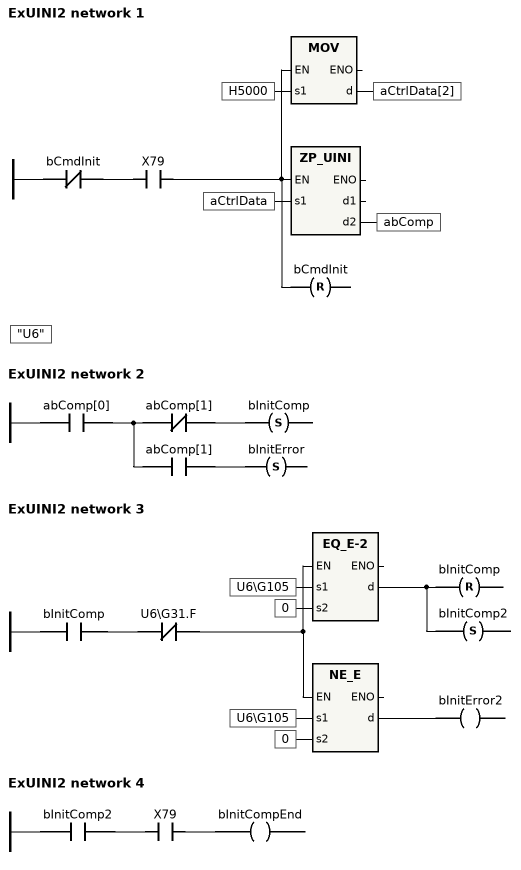
(* [picture p48: structured ladder/FBD of ExUINI2, networks 1 to 4] *)
(* network 1 *)
_p1 := NOT bCmdInit AND X79;
MOV(_p1, H5000, aCtrlData[2]);
ZP_UINI(_p1, aCtrlData, _open, abComp);
RST(_p1, bCmdInit);
(* not connected to any output: "U6" *)
(* network 2 *)
SET(abComp[0] AND NOT abComp[1], bInitComp);
SET(abComp[0] AND abComp[1], bInitError);
(* network 3 *)
_p1 := bInitComp AND NOT U6\G31.F;
EQ_E(_p1, U6\G105, 0, _t2);
RST(_t2, bInitComp);
SET(_t2, bInitComp2);
NE_E(_p1, U6\G105, 0, _t3);
bInitError2 := _t3;
(* network 4 *)
bInitCompEnd := bInitComp2 AND X79;
END_PROGRAM

PROGRAM ExEthSREAD_SWRITE
VAR
  Mov8INT_1 : Mov8INT;
  acRdCtrl : ARRAY [0..17] OF INT;
  abRdComp : ARRAY [0..1] OF BOOL;
  iCntRdOk : INT;
  iCntRdErr : INT;
  acWrCtrl : ARRAY [0..17] OF INT;
  abWrComp : ARRAY [0..1] OF BOOL;
  Mov8INT_2 : Mov8INT;
  iCntWrOk : INT;
  iCntWrErr : INT;
  bRdOK : BOOL;
  bWrOK : BOOL;
END_VAR
(* structured ladder/FBD written out as ST: instructions are called as NAME(EN, inputs, outputs); _pN, _eN, _tN stand for wires *)
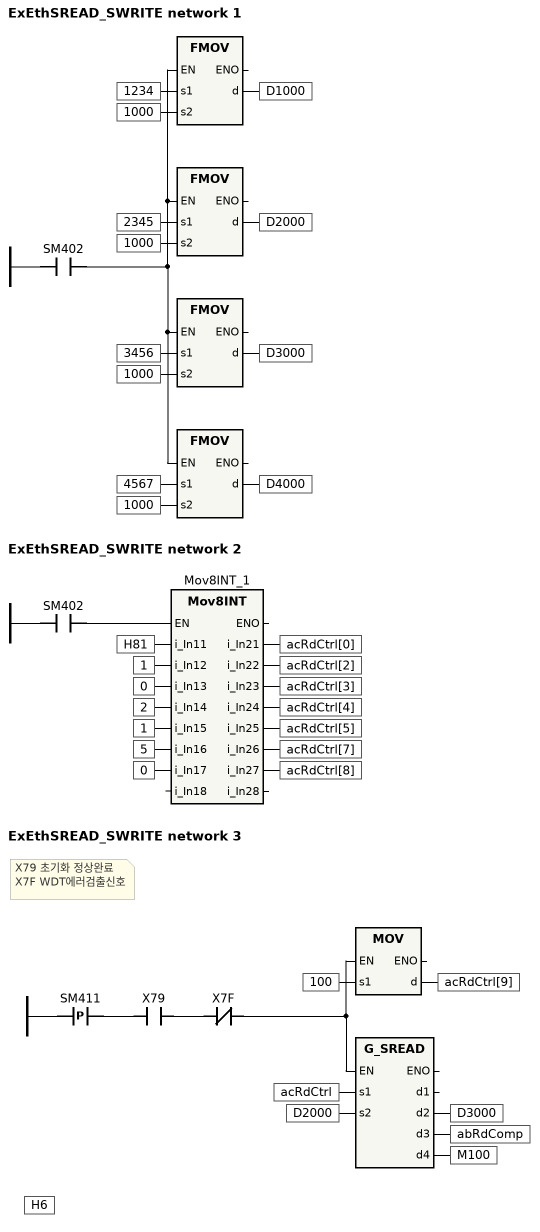
(* network 1 *)
FMOV(SM402, 1234, 1000, D1000);
FMOV(SM402, 2345, 1000, D2000);
FMOV(SM402, 3456, 1000, D3000);
FMOV(SM402, 4567, 1000, D4000);
(* network 2 *)
Mov8INT_1(EN := SM402, i_In11 := H81, i_In12 := 1, i_In13 := 0, i_In14 := 2, i_In15 := 1, i_In16 := 5, i_In17 := 0, i_In21 => acRdCtrl[0], i_In22 => acRdCtrl[2], i_In23 => acRdCtrl[3], i_In24 => acRdCtrl[4], i_In25 => acRdCtrl[5], i_In26 => acRdCtrl[7], i_In27 => acRdCtrl[8]);
(* network 3 *)
(* X79 초기화 정상완료 / X7F WDT에러검출신호 *)
_p1 := LDP(TRUE, SM411) AND X79 AND NOT X7F;
MOV(_p1, 100, acRdCtrl[9]);
G_SREAD(_p1, acRdCtrl, D2000, _open, D3000, abRdComp, M100);
(* not connected to any output: H6 *)
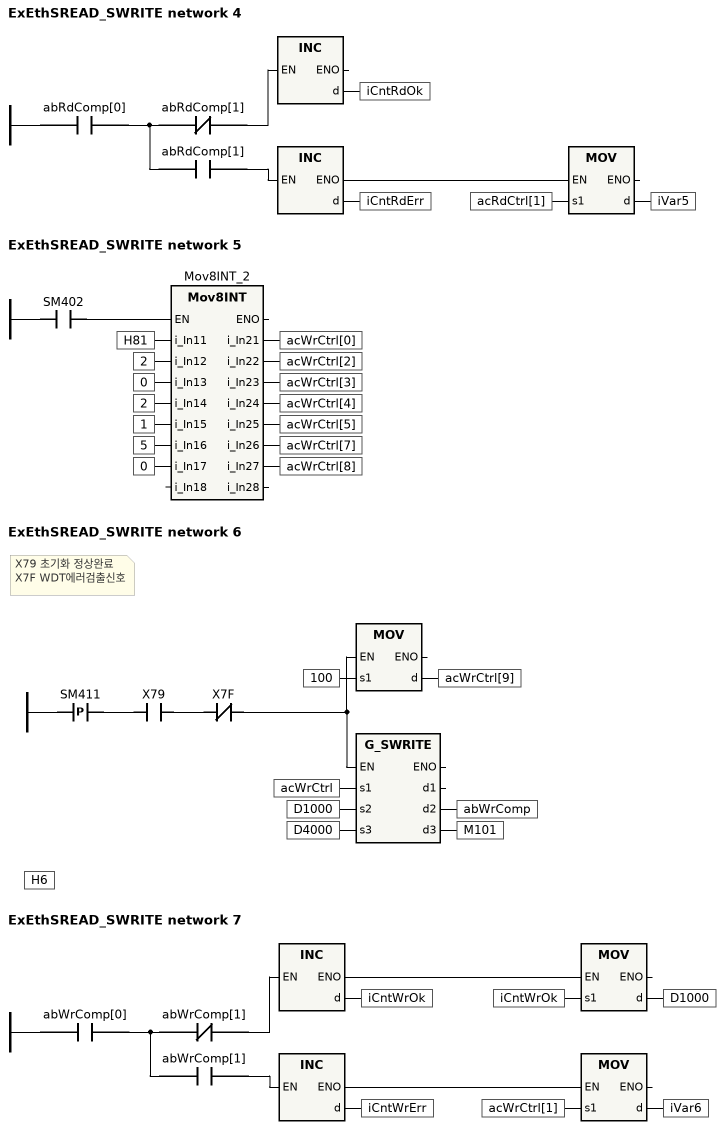
(* network 4 *)
INC(abRdComp[0] AND NOT abRdComp[1], iCntRdOk);
_e1 := INC(abRdComp[0] AND abRdComp[1], iCntRdErr);
MOV(_e1, acRdCtrl[1], iVar5);
(* network 5 *)
Mov8INT_2(EN := SM402, i_In11 := H81, i_In12 := 2, i_In13 := 0, i_In14 := 2, i_In15 := 1, i_In16 := 5, i_In17 := 0, i_In21 => acWrCtrl[0], i_In22 => acWrCtrl[2], i_In23 => acWrCtrl[3], i_In24 => acWrCtrl[4], i_In25 => acWrCtrl[5], i_In26 => acWrCtrl[7], i_In27 => acWrCtrl[8]);
(* network 6 *)
(* X79 초기화 정상완료 / X7F WDT에러검출신호 *)
_p1 := LDP(TRUE, SM411) AND X79 AND NOT X7F;
MOV(_p1, 100, acWrCtrl[9]);
G_SWRITE(_p1, acWrCtrl, D1000, D4000, _open, abWrComp, M101);
(* not connected to any output: H6 *)
(* network 7 *)
_e1 := INC(abWrComp[0] AND NOT abWrComp[1], iCntWrOk);
MOV(_e1, iCntWrOk, D1000);
_e2 := INC(abWrComp[0] AND abWrComp[1], iCntWrErr);
MOV(_e2, acWrCtrl[1], iVar6);
END_PROGRAM

PROGRAM ExREQ
VAR
  Mov8INT_1 : Mov8INT;
  acReqCtrl : ARRAY [0..17] OF INT;
  abReqComp : ARRAY [0..1] OF BOOL;
  aReqData : ARRAY [0..5] OF INT;
  Mov8INT_2 : Mov8INT;
  aAnsData : ARRAY [0..5] OF INT;
  Mov4INT_1 : Mov4INT;
  ReqCmd : BOOL;
  iCntReqOk : INT;
  iCntReqErr : INT;
  ReqClock : BOOL;
  acClkCtrl : ARRAY [0..17] OF INT;
  abClkComp : ARRAY [0..1] OF BOOL;
  iCntClkOk : INT;
  iCntClkErr : INT;
  Mov4INT_2 : Mov4INT;
  aClkData : ARRAY [0..5] OF INT;
  Mov4INT_3 : Mov4INT;
  Mov4INT_4 : Mov4INT;
END_VAR
(* structured ladder/FBD written out as ST: instructions are called as NAME(EN, inputs, outputs); _pN, _eN, _tN stand for wires *)
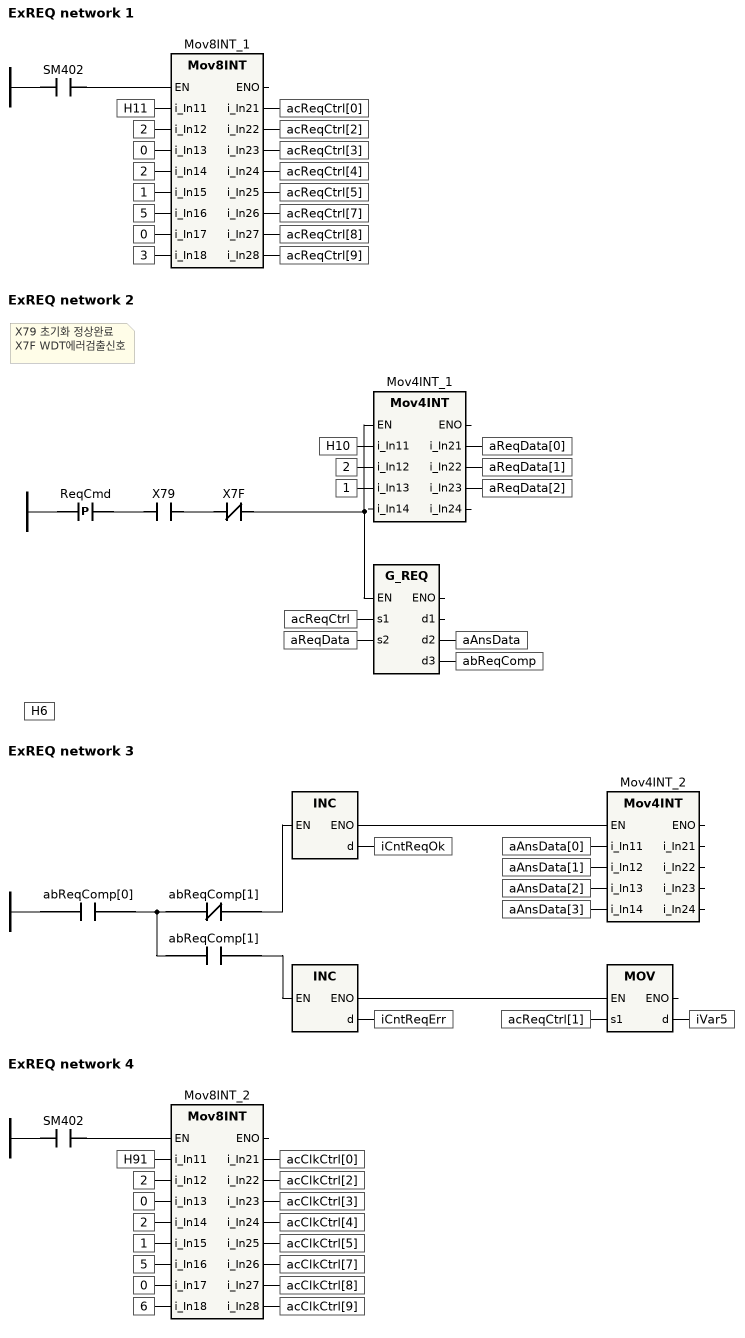
(* network 1 *)
Mov8INT_1(EN := SM402, i_In11 := H11, i_In12 := 2, i_In13 := 0, i_In14 := 2, i_In15 := 1, i_In16 := 5, i_In17 := 0, i_In18 := 3, i_In21 => acReqCtrl[0], i_In22 => acReqCtrl[2], i_In23 => acReqCtrl[3], i_In24 => acReqCtrl[4], i_In25 => acReqCtrl[5], i_In26 => acReqCtrl[7], i_In27 => acReqCtrl[8], i_In28 => acReqCtrl[9]);
(* network 2 *)
(* X79 초기화 정상완료 / X7F WDT에러검출신호 *)
_p1 := LDP(TRUE, ReqCmd) AND X79 AND NOT X7F;
Mov4INT_1(EN := _p1, i_In11 := H10, i_In12 := 2, i_In13 := 1, i_In21 => aReqData[0], i_In22 => aReqData[1], i_In23 => aReqData[2]);
G_REQ(_p1, acReqCtrl, aReqData, _open, aAnsData, abReqComp);
(* not connected to any output: H6 *)
(* network 3 *)
_e1 := INC(abReqComp[0] AND NOT abReqComp[1], iCntReqOk);
Mov4INT_2(EN := _e1, i_In11 := aAnsData[0], i_In12 := aAnsData[1], i_In13 := aAnsData[2], i_In14 := aAnsData[3]);
_e2 := INC(abReqComp[0] AND abReqComp[1], iCntReqErr);
MOV(_e2, acReqCtrl[1], iVar5);
(* network 4 *)
Mov8INT_2(EN := SM402, i_In11 := H91, i_In12 := 2, i_In13 := 0, i_In14 := 2, i_In15 := 1, i_In16 := 5, i_In17 := 0, i_In18 := 6, i_In21 => acClkCtrl[0], i_In22 => acClkCtrl[2], i_In23 => acClkCtrl[3], i_In24 => acClkCtrl[4], i_In25 => acClkCtrl[5], i_In26 => acClkCtrl[7], i_In27 => acClkCtrl[8], i_In28 => acClkCtrl[9]);
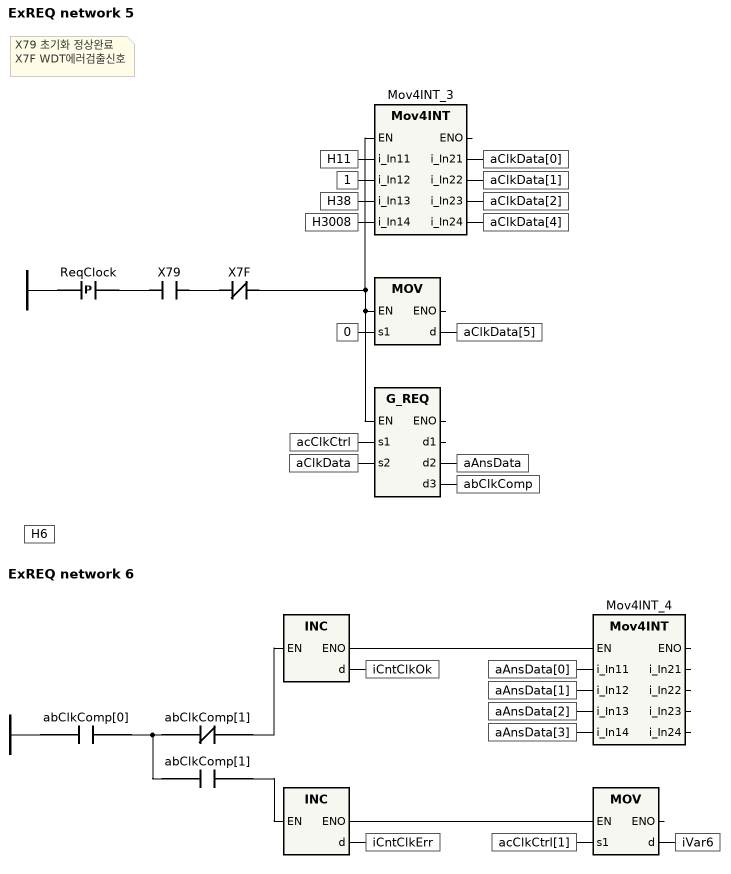
(* network 5 *)
(* X79 초기화 정상완료 / X7F WDT에러검출신호 *)
_p1 := LDP(TRUE, ReqClock) AND X79 AND NOT X7F;
Mov4INT_3(EN := _p1, i_In11 := H11, i_In12 := 1, i_In13 := H38, i_In14 := H3008, i_In21 => aClkData[0], i_In22 => aClkData[1], i_In23 => aClkData[2], i_In24 => aClkData[4]);
MOV(_p1, 0, aClkData[5]);
G_REQ(_p1, acClkCtrl, aClkData, _open, aAnsData, abClkComp);
(* not connected to any output: H6 *)
(* network 6 *)
_e1 := INC(abClkComp[0] AND NOT abClkComp[1], iCntClkOk);
Mov4INT_4(EN := _e1, i_In11 := aAnsData[0], i_In12 := aAnsData[1], i_In13 := aAnsData[2], i_In14 := aAnsData[3]);
_e2 := INC(abClkComp[0] AND abClkComp[1], iCntClkErr);
MOV(_e2, acClkCtrl[1], iVar6);
END_PROGRAM

PROGRAM ExSEND_RECV
VAR
  Mov8INT_1 : Mov8INT;
  acSndCtrl : ARRAY [0..17] OF INT;
  abSndComp : ARRAY [0..1] OF BOOL;
  aSndData : ARRAY [0..3] OF INT;
  Mov8INT_2 : Mov8INT;
  aAnsData : ARRAY [0..5] OF INT;
  Mov4INT_1 : Mov4INT;
  iCntSndOk : INT;
  iCntSndErr : INT;
  acRevCtrl : ARRAY [0..17] OF INT;
  abRevComp : ARRAY [0..1] OF BOOL;
  iCntRevOk : INT;
  iCntRevErr : INT;
  Mov4INT_2 : Mov4INT;
  aRevData : ARRAY [0..3] OF INT;
  Mov4INT_3 : Mov4INT;
  Mov4INT_4 : Mov4INT;
  SendCmd : BOOL;
  RecvCmd : BOOL;
END_VAR
(* structured ladder/FBD written out as ST: instructions are called as NAME(EN, inputs, outputs); _pN, _eN, _tN stand for wires *)
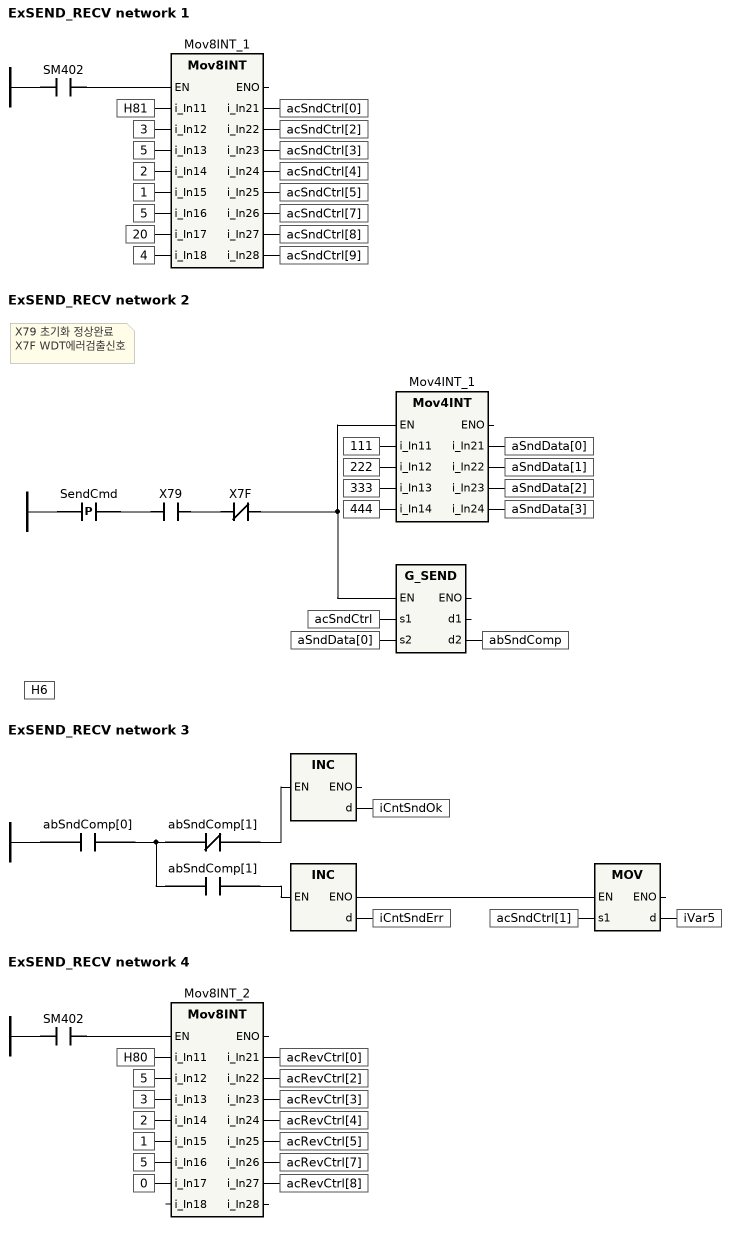
(* network 1 *)
Mov8INT_1(EN := SM402, i_In11 := H81, i_In12 := 3, i_In13 := 5, i_In14 := 2, i_In15 := 1, i_In16 := 5, i_In17 := 20, i_In18 := 4, i_In21 => acSndCtrl[0], i_In22 => acSndCtrl[2], i_In23 => acSndCtrl[3], i_In24 => acSndCtrl[4], i_In25 => acSndCtrl[5], i_In26 => acSndCtrl[7], i_In27 => acSndCtrl[8], i_In28 => acSndCtrl[9]);
(* network 2 *)
(* X79 초기화 정상완료 / X7F WDT에러검출신호 *)
_p1 := LDP(TRUE, SendCmd) AND X79 AND NOT X7F;
Mov4INT_1(EN := _p1, i_In11 := 111, i_In12 := 222, i_In13 := 333, i_In14 := 444, i_In21 => aSndData[0], i_In22 => aSndData[1], i_In23 => aSndData[2], i_In24 => aSndData[3]);
G_SEND(_p1, acSndCtrl, aSndData[0], _open, abSndComp);
(* not connected to any output: H6 *)
(* network 3 *)
INC(abSndComp[0] AND NOT abSndComp[1], iCntSndOk);
_e1 := INC(abSndComp[0] AND abSndComp[1], iCntSndErr);
MOV(_e1, acSndCtrl[1], iVar5);
(* network 4 *)
Mov8INT_2(EN := SM402, i_In11 := H80, i_In12 := 5, i_In13 := 3, i_In14 := 2, i_In15 := 1, i_In16 := 5, i_In17 := 0, i_In21 => acRevCtrl[0], i_In22 => acRevCtrl[2], i_In23 => acRevCtrl[3], i_In24 => acRevCtrl[4], i_In25 => acRevCtrl[5], i_In26 => acRevCtrl[7], i_In27 => acRevCtrl[8]);
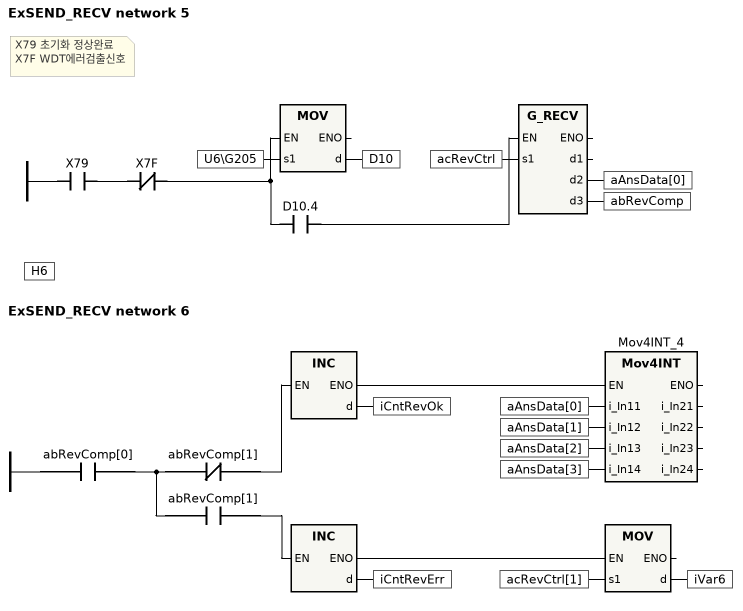
(* network 5 *)
(* X79 초기화 정상완료 / X7F WDT에러검출신호 *)
_p1 := X79 AND NOT X7F;
MOV(_p1, U6\G205, D10);
G_RECV(_p1 AND D10.4, acRevCtrl, _open, aAnsData[0], abRevComp);
(* not connected to any output: H6 *)
(* network 6 *)
_e1 := INC(abRevComp[0] AND NOT abRevComp[1], iCntRevOk);
Mov4INT_4(EN := _e1, i_In11 := aAnsData[0], i_In12 := aAnsData[1], i_In13 := aAnsData[2], i_In14 := aAnsData[3]);
_e2 := INC(abRevComp[0] AND abRevComp[1], iCntRevErr);
MOV(_e2, acRevCtrl[1], iVar6);
END_PROGRAM

PROGRAM ExRECVS_INT
VAR
  acRevCtrl : ARRAY [0..17] OF INT;
  abRevComp : ARRAY [0..1] OF BOOL;
  iCntRevOk : INT;
END_VAR
(* structured ladder/FBD written out as ST: instructions are called as NAME(EN, inputs, outputs); _pN, _eN, _tN stand for wires *)
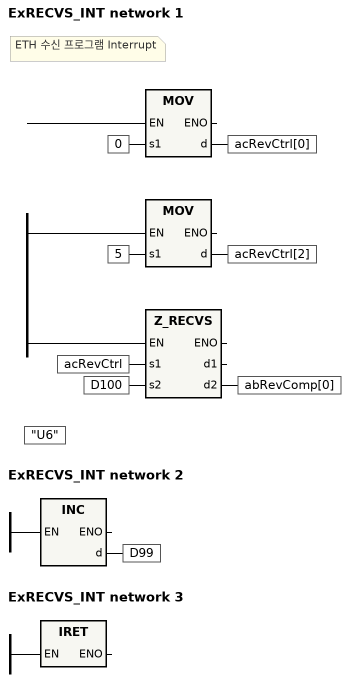
(* network 1 *)
(* ETH 수신 프로그램 Interrupt *)
MOV(TRUE, 0, acRevCtrl[0]);
MOV(TRUE, 5, acRevCtrl[2]);
Z_RECVS(TRUE, acRevCtrl, D100, _open, abRevComp[0]);
(* not connected to any output: "U6" *)
(* network 2 *)
INC(TRUE, D99);
(* network 3 *)
IRET(TRUE);
END_PROGRAM

PROGRAM ExRECVS
VAR
  Mov8INT_1 : Mov8INT;
  Mov8INT_2 : Mov8INT;
END_VAR
(* structured ladder/FBD written out as ST: instructions are called as NAME(EN, inputs, outputs); _pN, _eN, _tN stand for wires *)
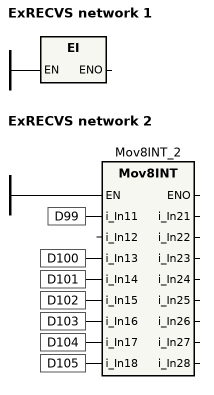
(* network 1 *)
EI(TRUE);
(* network 2 *)
Mov8INT_2(EN := TRUE, i_In11 := D99, i_In13 := D100, i_In14 := D101, i_In15 := D102, i_In16 := D103, i_In17 := D104, i_In18 := D105);
END_PROGRAM

PROGRAM ExZNRD_ZNWR
VAR
  Mov8INT_1 : Mov8INT;
  acRdCtrl : ARRAY [0..17] OF INT;
  abRdComp : ARRAY [0..1] OF BOOL;
  iCntRdOk : INT;
  iCntRdErr : INT;
  acWrCtrl : ARRAY [0..17] OF INT;
  abWrComp : ARRAY [0..1] OF BOOL;
  Mov8INT_2 : Mov8INT;
  iCntWrOk : INT;
  iCntWrErr : INT;
END_VAR
(* structured ladder/FBD written out as ST: instructions are called as NAME(EN, inputs, outputs); _pN, _eN, _tN stand for wires *)
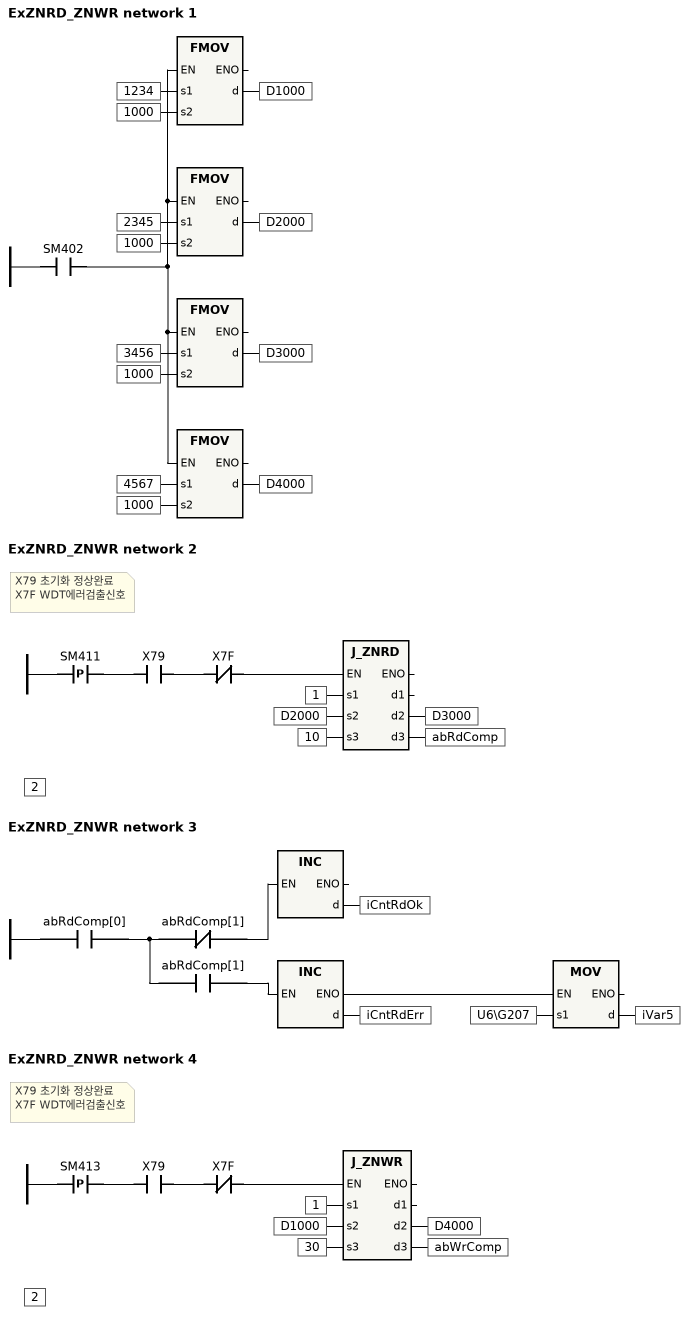
(* network 1 *)
FMOV(SM402, 1234, 1000, D1000);
FMOV(SM402, 2345, 1000, D2000);
FMOV(SM402, 3456, 1000, D3000);
FMOV(SM402, 4567, 1000, D4000);
(* network 2 *)
(* X79 초기화 정상완료 / X7F WDT에러검출신호 *)
J_ZNRD(LDP(TRUE, SM411) AND X79 AND NOT X7F, 1, D2000, 10, _open, D3000, abRdComp);
(* not connected to any output: 2 *)
(* network 3 *)
INC(abRdComp[0] AND NOT abRdComp[1], iCntRdOk);
_e1 := INC(abRdComp[0] AND abRdComp[1], iCntRdErr);
MOV(_e1, U6\G207, iVar5);
(* network 4 *)
(* X79 초기화 정상완료 / X7F WDT에러검출신호 *)
J_ZNWR(LDP(TRUE, SM413) AND X79 AND NOT X7F, 1, D1000, 30, _open, D4000, abWrComp);
(* not connected to any output: 2 *)
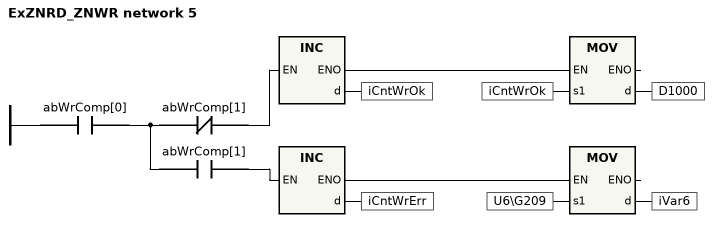
(* network 5 *)
_e1 := INC(abWrComp[0] AND NOT abWrComp[1], iCntWrOk);
MOV(_e1, iCntWrOk, D1000);
_e2 := INC(abWrComp[0] AND abWrComp[1], iCntWrErr);
MOV(_e2, U6\G209, iVar6);
END_PROGRAM

PROGRAM ExMSEND2
VAR
  abComp : ARRAY [0..1] OF BOOL;
  Mov4INT_1 : Mov4INT;
  aCtrlData : ARRAY [0..15] OF INT;
  bCmdFlag : BOOL;
  bExeFlag : BOOL;
  Mov4INT_2 : Mov4INT;
END_VAR
(* structured ladder/FBD written out as ST: instructions are called as NAME(EN, inputs, outputs); _pN, _eN, _tN stand for wires *)
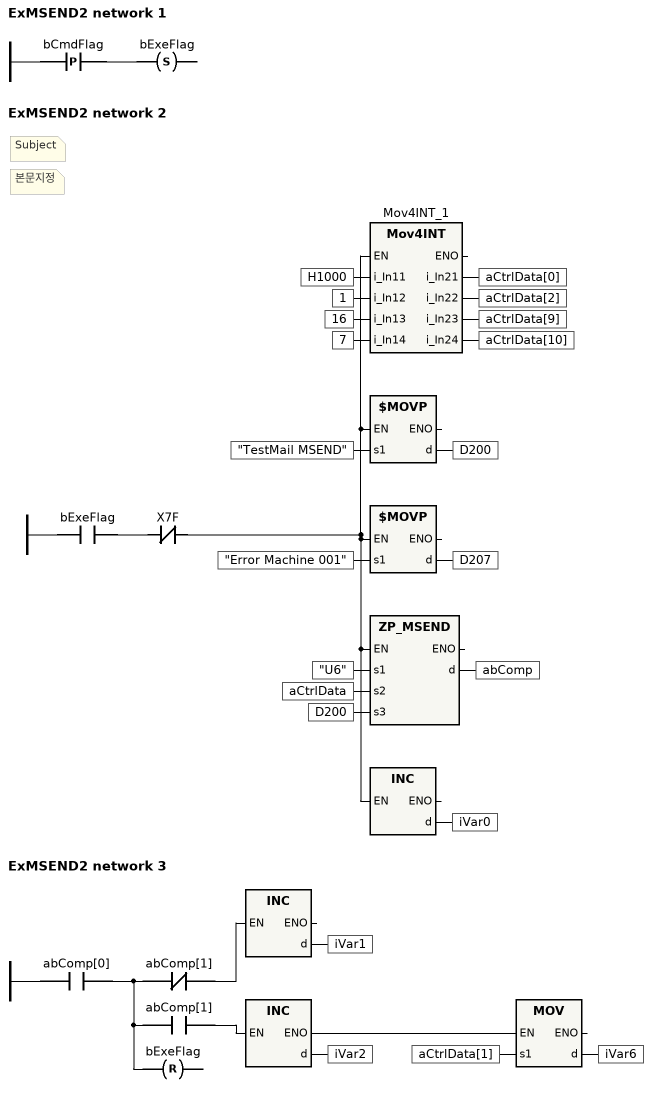
(* network 1 *)
SET(LDP(TRUE, bCmdFlag), bExeFlag);
(* network 2 *)
(* Subject *)
(* 본문지정 *)
_p1 := bExeFlag AND NOT X7F;
Mov4INT_1(EN := _p1, i_In11 := H1000, i_In12 := 1, i_In13 := 16, i_In14 := 7, i_In21 => aCtrlData[0], i_In22 => aCtrlData[2], i_In23 => aCtrlData[9], i_In24 => aCtrlData[10]);
$MOVP(_p1, "TestMail MSEND", D200);
$MOVP(_p1, "Error Machine 001", D207);
ZP_MSEND(_p1, "U6", aCtrlData, D200, abComp);
INC(_p1, iVar0);
(* network 3 *)
INC(abComp[0] AND NOT abComp[1], iVar1);
_e1 := INC(abComp[0] AND abComp[1], iVar2);
MOV(_e1, aCtrlData[1], iVar6);
RST(abComp[0], bExeFlag);
END_PROGRAM

PROGRAM ExECPRTCL
VAR
  bModeReq : BOOL;
  bCmdReq : BOOL;
  abRes : ARRAY [0..1] OF BOOL;
  bOK : BOOL;
  bERR : BOOL;
  Mov8INT_2 : Mov8INT;
  Word2Bit16_1 : Word2Bit16;
  Word2Bit16_2 : Word2Bit16;
  Word2Bit16_3 : Word2Bit16;
  Mov8INT_1 : Mov8INT;
  Mov8INT_3 : Mov8INT;
END_VAR
(* structured ladder/FBD written out as ST: instructions are called as NAME(EN, inputs, outputs); _pN, _eN, _tN stand for wires *)
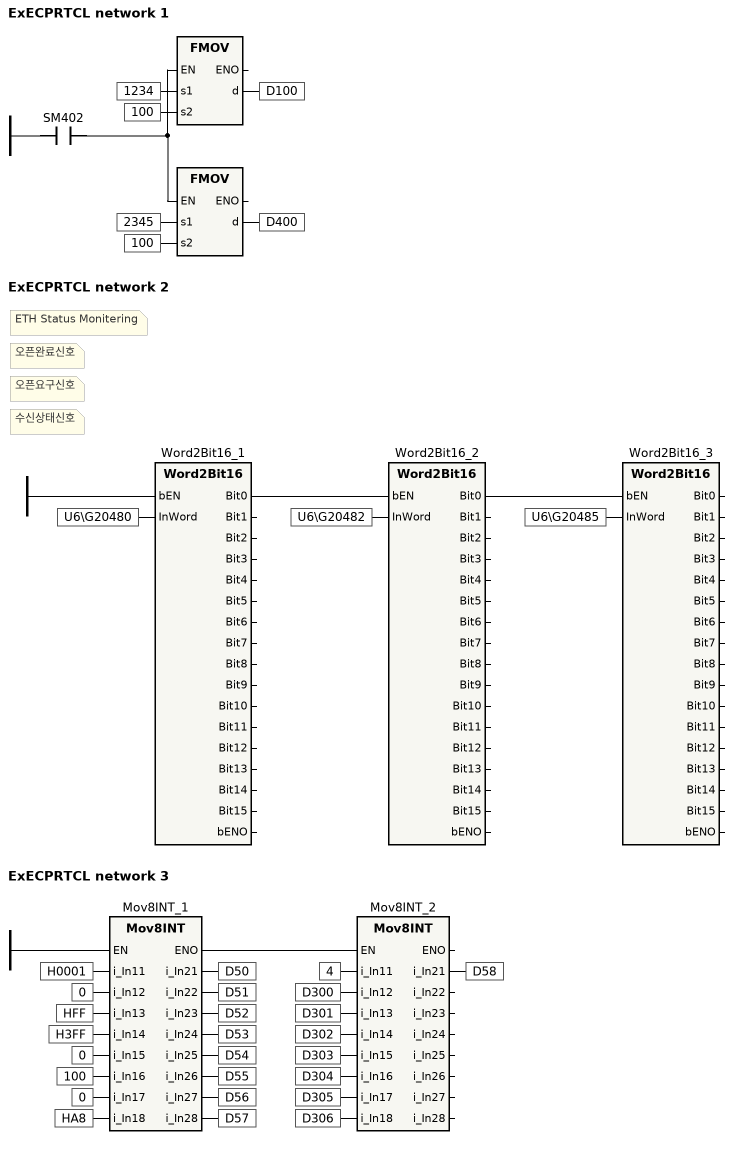
(* network 1 *)
FMOV(SM402, 1234, 100, D100);
FMOV(SM402, 2345, 100, D400);
(* network 2 *)
(* ETH Status Monitering *)
(* 오픈완료신호 *)
(* 오픈요구신호 *)
(* 수신상태신호 *)
Word2Bit16_1(bEN := TRUE, InWord := U6\G20480);
Word2Bit16_2(bEN := Word2Bit16_1.Bit0, InWord := U6\G20482);
Word2Bit16_3(bEN := Word2Bit16_2.Bit0, InWord := U6\G20485);
(* network 3 *)
Mov8INT_1(EN := TRUE, i_In11 := H0001, i_In12 := 0, i_In13 := HFF, i_In14 := H3FF, i_In15 := 0, i_In16 := 100, i_In17 := 0, i_In18 := HA8, i_In21 => D50, i_In22 => D51, i_In23 => D52, i_In24 => D53, i_In25 => D54, i_In26 => D55, i_In27 => D56, i_In28 => D57);
Mov8INT_2(EN := Mov8INT_1.ENO, i_In11 := 4, i_In12 := D300, i_In13 := D301, i_In14 := D302, i_In15 := D303, i_In16 := D304, i_In17 := D305, i_In18 := D306, i_In21 => D58);
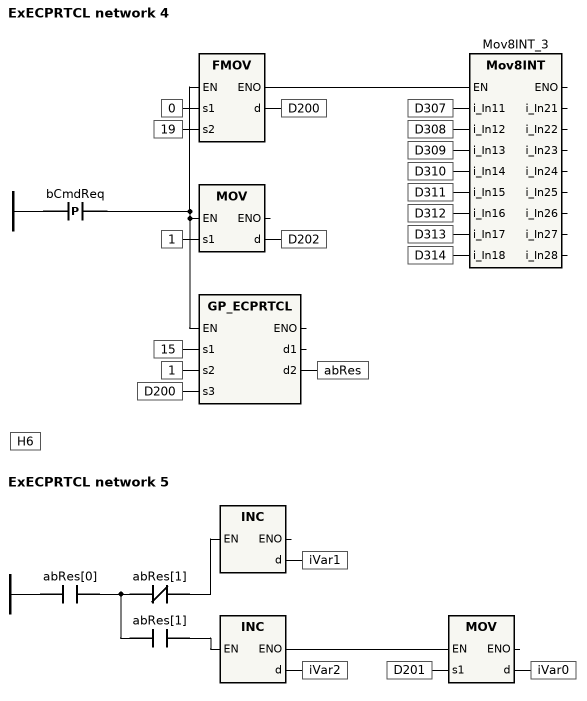
(* network 4 *)
_p1 := LDP(TRUE, bCmdReq);
_e2 := FMOV(_p1, 0, 19, D200);
Mov8INT_3(EN := _e2, i_In11 := D307, i_In12 := D308, i_In13 := D309, i_In14 := D310, i_In15 := D311, i_In16 := D312, i_In17 := D313, i_In18 := D314);
MOV(_p1, 1, D202);
GP_ECPRTCL(_p1, 15, 1, D200, _open, abRes);
(* not connected to any output: H6 *)
(* network 5 *)
INC(abRes[0] AND NOT abRes[1], iVar1);
_e1 := INC(abRes[0] AND abRes[1], iVar2);
MOV(_e1, D201, iVar0);
END_PROGRAM
